// TIA Portal V21 export
VAR_GLOBAL   // PLC tag table "KAllZona"
END_VAR
VAR_GLOBAL CONSTANT   // user constants
   KAllZone_CentralinaSicurezza : Int := 1;
   KAllZone_PressostatoGenerale : Int := 3;
   KAllZone_CicloNonInserito : Int := 2;
END_VAR
